(* CoDeSys 2.3.9.41 project: VOS_Vorkuta_ASU_1.pro *)
(* Libraries: GermesLib_1_51.lib 19.5.21 13:36:15, PID_Regulators.lib 6.11.19 15:29:27, Util.lib 18.5.10 15:14:28, STANDARD.LIB 4.10.05 11:14:46, IECSFC.LIB 13.4.06 15:51:28, SYSLIBTIME.LIB 6.11.19 15:29:28, ANALYZATION.LIB 5.10.99 09:05:06 *)

(* PLC configuration (modules and I/O channels)
Fast discrete inputs [I_SIMPLE_INPUT] node 0, in %IB0 out %QB0 {ChannellName = Fast discrete inputs; Filtrationtime = 10000}
  DD1_DI_1 AT %IX0.0 [BitInput] Discrete input 1 reserve {ChannellName = Enter name}
  DD1_DI_2 AT %IX0.1 [BitInput] Discrete input 2 reserve {ChannellName = Enter name}
  DD1_DI_3 AT %IX0.2 [BitInput] Discrete input 3 reserve {ChannellName = Enter name}
  DD1_DI_4 AT %IX0.3 [BitInput] Discrete input 4 reserve {ChannellName = Enter name}
Discrete inputs [ID130] node 1, in %IB1 out %QB1 {ChannellName = Discrete inputs; Filtrationtime_GeneralINP = 10; PinCount = 12; Visibility = No}
  AT %IB1.0 [ByteInput] 8 discrete inputs {ChannellName = Enter name}
  AT %IB1.1 [ByteInput] 4 discrete inputs {ChannellName = Enter name}
Fast discrete outputs [OWEN_ID570] node 2, in %IB2 out %QB2 {ChannellName = Fast discrete outputs; SafeValueBool = FALSE; SafeValueBool = FALSE; SafeValueBool = FALSE; SafeValueBool = FALSE; Visibility = No}
  AT %QX2.0 [BitOutput] Fast discrete output 1 {ChannellName = Enter name}
  AT %QX2.1 [BitOutput] Fast discrete output 2 {ChannellName = Enter name}
  AT %QX2.2 [BitOutput] Fast discrete output 3 {ChannellName = Enter name}
  AT %QX2.3 [BitOutput] Fast discrete output 4 {ChannellName = Enter name}
Discrete outputs [ID131] node 3, in %IB3 out %QB3 {ChannellName = Discrete outputs; SafeValueByte = 0; Visibility = No}
  AT %QB3.0 [ByteOutput] 8 discrete outputs {ChannellName = Enter name}
  AT %QB3.1 [ByteOutput] 8 discrete outputs {ChannellName = Enter name}
DD1_AI_1 AT %IR4.0 [FloatInputP] LT06.01/01 уровень в V06.01/01 {ChannellName = Fast analog input; AIN_TYPE = 0-20 mA; Peak_Filtr = 200; Flt_Ch = Off; TauRC = 10; MinFV = 0; MaxFV = 20000.0}
DD1_AI_2 AT %IR4.1 [FloatInputP] PT06.01/01 {ChannellName = Fast analog input; AIN_TYPE = 0-20 mA; Peak_Filtr = 200; Flt_Ch = Off; TauRC = 10; MinFV = 0; MaxFV = 20000.0}
DD1_AI_3 AT %IR4.2 [FloatInputP] PT06.01/02 {ChannellName = Fast analog input; AIN_TYPE = 0-20 mA; Peak_Filtr = 200; Flt_Ch = Off; TauRC = 10; MinFV = 0; MaxFV = 20000.0}
DD1_AI_4 AT %IR4.3 [FloatInputP] TT01.02 температура воздуха в помещении {ChannellName = Fast analog input; AIN_TYPE = 0-20 mA; Peak_Filtr = 200; Flt_Ch = Off; TauRC = 10; MinFV = 0; MaxFV = 20000.0}
DD1_AI_5 AT %IR4.4 [FloatInputP] TT06.01 температура воды на выходе {ChannellName = Fast analog input; AIN_TYPE = 0-20 mA; Peak_Filtr = 200; Flt_Ch = Off; TauRC = 10; MinFV = 0; MaxFV = 20000.0}
DD1_AI_6 AT %IR4.5 [FloatInputP] pH-метр QE06.01 {ChannellName = Fast analog input; AIN_TYPE = 0-20 mA; Peak_Filtr = 200; Flt_Ch = Off; TauRC = 10; MinFV = 0; MaxFV = 20000.0}
DD1_AI_7 AT %IR4.6 [FloatInputP] FIT06.01 расходомер на выходе {ChannellName = Fast analog input; AIN_TYPE = 0-20 mA; Peak_Filtr = 200; Flt_Ch = Off; TauRC = 10; MinFV = 0; MaxFV = 20000.0}
DD1_AI_8 AT %IR4.7 [FloatInputP] reserve {ChannellName = Fast analog input; AIN_TYPE = 0-20 mA; Peak_Filtr = 200; Flt_Ch = Off; TauRC = 10; MinFV = 0; MaxFV = 20000.0}
AT %IW4.8 [WordInput] AI read time (10ms) {ChannellName = Enter name}
Analog outputs [ID126] node 5, in %IB5 out %QB5 {ChannellName = Analog outputs}
  DD1_AO_1 AT %QR5.0 [FloatOutputP] производительность доз.насоса Р03.06/01 {ChannellName = Analog output; AOUT_TYPE = 4-20 mA; SafeValueREAL = 0.0}
  DD1_AO_2 AT %QR5.1 [FloatOutputP] производительность доз.насоса Р03.06/02 {ChannellName = Analog output; AOUT_TYPE = 4-20 mA; SafeValueREAL = 0.0}
  DD1_AO_3 AT %QR5.2 [FloatOutputP] reserve {ChannellName = Analog output; AOUT_TYPE = 4-20 mA; SafeValueREAL = 0.0}
  DD1_AO_4 AT %QR5.3 [FloatOutputP] reserve {ChannellName = Analog output; AOUT_TYPE = 4-20 mA; SafeValueREAL = 0.0}
Special input [ID103] node 6, in %IB6 out %QB6 {ChannellName = Special input}
  AT %IX6.0 [BitInput] Special input {ChannellName = Enter name}
Special output [ID104] node 7, in %IB7 out %QB7 {ChannellName = Special output}
  AT %QX7.0 [BitOutput] Special output {ChannellName = Enter name}
AT %QD8.0 [DWordOutput] Last address {ChannellName = Enter name}
AT %QW8.1 [WordOutput] Last error {ChannellName = Enter name}
RS-485-1 [COM1_USART] node 0, in %IB8.0 out %QB8.0 {ChannellName = RS-485-1; CommunicationSpeed = 115200; Parity = NO PARITY CHECK; BitLength = 8 bits; StopLength = One stop bit; InterfaceType = RS485; FrameOriented = RTU; Timeout = 2; Visibility = No}
Universal Modbus device [ID2000] node 1, in %IB8.1 out %QB8.1 {ChannellName = Universal Modbus device; ModuleIP = 10:0:0:223; ServiceTimeout = 150; TCPport = 502; NetMode = Serial; ModuleSlaveAddress = 11; RequestType = By poll time; PeriodOfService = 100; Visibility = No; RepeatCounter = 0; ByteSequence = Native}
  AT %QB8.1.0 [ComChannel] Command (0xff - Start) {ChannellName = Enter name}
  Real input module [ID2007] node 0, in %IB8.1.0 out %QB8.1.0 {ChannellName = float input module; ModbusAddress = 512; Command_read_regs = Read holding Registers  (0x03); Visibility = No}
    DD2_AI_1 AT %QD8.1.0.0 [FloatOutput] {ChannellName = Enter name}
  Real input module [ID2007] node 1, in %IB8.1.1 out %QB8.1.1 {ChannellName = float input module; ModbusAddress = 514; Command_read_regs = Read holding Registers  (0x03); Visibility = No}
    DD2_AI_2 AT %QD8.1.1.0 [FloatOutput] {ChannellName = Enter name}
  Real input module [ID2007] node 2, in %IB8.1.2 out %QB8.1.2 {ChannellName = float input module; ModbusAddress = 516; Command_read_regs = Read holding Registers  (0x03); Visibility = No}
    DD2_AI_3 AT %QD8.1.2.0 [FloatOutput] {ChannellName = Enter name}
  Real input module [ID2007] node 3, in %IB8.1.3 out %QB8.1.3 {ChannellName = float input module; ModbusAddress = 518; Command_read_regs = Read holding Registers  (0x03); Visibility = No}
    DD2_AI_4 AT %QD8.1.3.0 [FloatOutput] {ChannellName = Enter name}
  Real input module [ID2007] node 4, in %IB8.1.4 out %QB8.1.4 {ChannellName = float input module; ModbusAddress = 520; Command_read_regs = Read holding Registers  (0x03); Visibility = No}
    DD2_AI_5 AT %QD8.1.4.0 [FloatOutput] {ChannellName = Enter name}
  Real input module [ID2007] node 5, in %IB8.1.5 out %QB8.1.5 {ChannellName = float input module; ModbusAddress = 522; Command_read_regs = Read holding Registers  (0x03); Visibility = No}
    DD2_AI_6 AT %QD8.1.5.0 [FloatOutput] {ChannellName = Enter name}
  Real input module [ID2007] node 6, in %IB8.1.6 out %QB8.1.6 {ChannellName = float input module; ModbusAddress = 524; Command_read_regs = Read holding Registers  (0x03); Visibility = No}
    DD2_AI_7 AT %QD8.1.6.0 [FloatOutput] {ChannellName = Enter name}
  Real input module [ID2007] node 7, in %IB8.1.7 out %QB8.1.7 {ChannellName = float input module; ModbusAddress = 526; Command_read_regs = Read holding Registers  (0x03); Visibility = No}
    DD2_AI_8 AT %QD8.1.7.0 [FloatOutput] {ChannellName = Enter name}
  Register input module [ID2003] node 8, in %IB8.1.8 out %QB8.1.8 {ChannellName = Register input module; ModbusAddress = 528; Command_read_regs = Read input registers  (0x04); Visibility = No}
    DI_BitMask AT %QW8.1.8.0 [WordOutput] {ChannellName = Enter name}
  Register input module [ID2003] node 9, in %IB8.1.9 out %QB8.1.9 {ChannellName = Register input module; ModbusAddress = 531; Command_read_regs = Read input registers  (0x04); Visibility = No}
    stat_word_PLC_DD2 AT %QW8.1.9.0 [WordOutput] {ChannellName = Enter name}
Universal Modbus device [ID2000] node 2, in %IB8.2 out %QB8.2 {ChannellName = Universal Modbus device; ModuleIP = 10:0:0:223; ServiceTimeout = 150; TCPport = 502; NetMode = Serial; ModuleSlaveAddress = 12; RequestType = By poll time; PeriodOfService = 100; Visibility = No; RepeatCounter = 0; ByteSequence = Native}
  AT %QB8.2.0 [ComChannel] Command (0xff - Start) {ChannellName = Enter name}
  Real input module [ID2007] node 0, in %IB8.2.0 out %QB8.2.0 {ChannellName = float input module; ModbusAddress = 512; Command_read_regs = Read holding Registers  (0x03); Visibility = No}
    DD3_AI_1 AT %QD8.2.0.0 [FloatOutput] {ChannellName = Enter name}
  Real input module [ID2007] node 1, in %IB8.2.1 out %QB8.2.1 {ChannellName = float input module; ModbusAddress = 514; Command_read_regs = Read holding Registers  (0x03); Visibility = No}
    DD3_AI_2 AT %QD8.2.1.0 [FloatOutput] {ChannellName = Enter name}
  Register input module [ID2003] node 2, in %IB8.2.2 out %QB8.2.2 {ChannellName = Register input module; ModbusAddress = 516; Command_read_regs = Read input registers  (0x04); Visibility = No}
    stat_word_PLC_DD3 AT %QW8.2.2.0 [WordOutput] {ChannellName = Enter name}
  Register input module [ID2003] node 3, in %IB8.2.3 out %QB8.2.3 {ChannellName = Register input module; ModbusAddress = 518; Command_read_regs = Read input registers  (0x04); Visibility = No}
    stat_ufo_PLC AT %QW8.2.3.0 [WordOutput] {ChannellName = Enter name}
Universal Modbus device [ID2000] node 3, in %IB8.3 out %QB8.3 {ChannellName = Universal Modbus device; ModuleIP = 10:0:0:223; ServiceTimeout = 150; TCPport = 502; NetMode = Serial; ModuleSlaveAddress = 13; RequestType = By poll time; PeriodOfService = 100; Visibility = No; RepeatCounter = 0; ByteSequence = Trace_mode}
  AT %QB8.3.0 [ComChannel] Command (0xff - Start) {ChannellName = Enter name}
  Register input module [ID2003] node 0, in %IB8.3.0 out %QB8.3.0 {ChannellName = Register input module; ModbusAddress = 17; Command_read_regs = Read input registers  (0x04); Visibility = No}
    bitMask_DD4_DI AT %QW8.3.0.0 [WordOutput] {ChannellName = Enter name}
Universal Modbus device [ID2000] node 4, in %IB8.4 out %QB8.4 {ChannellName = Universal Modbus device; ModuleIP = 10:0:0:223; ServiceTimeout = 150; TCPport = 502; NetMode = Serial; ModuleSlaveAddress = 11; RequestType = By value change; PeriodOfService = 100; Visibility = No; RepeatCounter = 0; ByteSequence = Native}
  AT %QB8.4.0 [ComChannel] Command (0xff - Start) {ChannellName = Enter name}
  Register output module State [ID2014] node 0, in %IB8.4.0 out %QB8.4.0 {ChannellName = Register output module State; ModbusAddress = 529; Command_write_one_reg = Write multiple registers(0x10); Visibility = No}
    DO_BitMask AT %QW8.4.0.0 [WordOutput] {ChannellName = Enter name}
    AT %QB8.4.0.1 [ComChannel] Command (0xff - Start) {ChannellName = Enter name}
  Register output module State [ID2014] node 1, in %IB8.4.1 out %QB8.4.1 {ChannellName = Register output module State; ModbusAddress = 530; Command_write_one_reg = Write multiple registers(0x10); Visibility = No}
    com_word_PLC_DD2 AT %QW8.4.1.0 [WordOutput] {ChannellName = Enter name}
    AT %QB8.4.1.1 [ComChannel] Command (0xff - Start) {ChannellName = Enter name}
  Register output module [ID2004] node 2, in %IB8.4.2 out %QB8.4.2 {ChannellName = Register; ModbusAddress = 532; Command_write_one_reg = Write multiple registers(0x10); Visibility = No}
    set_freq_p010301_PLC AT %QW8.4.2.0 [WordOutput] {ChannellName = Enter name}
  Register output module [ID2004] node 3, in %IB8.4.3 out %QB8.4.3 {ChannellName = Register; ModbusAddress = 533; Command_write_one_reg = Write multiple registers(0x10); Visibility = No}
    set_freq_p010302_PLC AT %QW8.4.3.0 [WordOutput] {ChannellName = Enter name}
  Register output module [ID2004] node 4, in %IB8.4.4 out %QB8.4.4 {ChannellName = Register; ModbusAddress = 534; Command_write_one_reg = Write multiple registers(0x10); Visibility = No}
    set_freq_p010303_PLC AT %QW8.4.4.0 [WordOutput] {ChannellName = Enter name}
  Register output module [ID2004] node 5, in %IB8.4.5 out %QB8.4.5 {ChannellName = Register; ModbusAddress = 535; Command_write_one_reg = Write multiple registers(0x10); Visibility = No}
    set_freq_p010701_PLC AT %QW8.4.5.0 [WordOutput] {ChannellName = Enter name}
  Register output module [ID2004] node 6, in %IB8.4.6 out %QB8.4.6 {ChannellName = Register; ModbusAddress = 536; Command_write_one_reg = Write multiple registers(0x10); Visibility = No}
    set_freq_p010702_PLC AT %QW8.4.6.0 [WordOutput] {ChannellName = Enter name}
  Register output module [ID2004] node 7, in %IB8.4.7 out %QB8.4.7 {ChannellName = Register; ModbusAddress = 537; Command_write_one_reg = Write multiple registers(0x10); Visibility = No}
    set_freq_p010801_PLC AT %QW8.4.7.0 [WordOutput] {ChannellName = Enter name}
  Register output module [ID2004] node 8, in %IB8.4.8 out %QB8.4.8 {ChannellName = Register; ModbusAddress = 538; Command_write_one_reg = Write multiple registers(0x10); Visibility = No}
    set_freq_p010802_PLC AT %QW8.4.8.0 [WordOutput] {ChannellName = Enter name}
  Register output module [ID2004] node 9, in %IB8.4.9 out %QB8.4.9 {ChannellName = Register; ModbusAddress = 539; Command_write_one_reg = Write multiple registers(0x10); Visibility = No}
    set_freq_p060201_PLC AT %QW8.4.9.0 [WordOutput] {ChannellName = Enter name}
  Register output module [ID2004] node 10, in %IB8.4.10 out %QB8.4.10 {ChannellName = Register; ModbusAddress = 540; Command_write_one_reg = Write multiple registers(0x10); Visibility = No}
    set_freq_p060202_PLC AT %QW8.4.10.0 [WordOutput] {ChannellName = Enter name}
Universal Modbus device [ID2000] node 5, in %IB8.5 out %QB8.5 {ChannellName = Universal Modbus device; ModuleIP = 10:0:0:223; ServiceTimeout = 150; TCPport = 502; NetMode = Serial; ModuleSlaveAddress = 12; RequestType = By value change; PeriodOfService = 100; Visibility = No; RepeatCounter = 0; ByteSequence = Native}
  AT %QB8.5.0 [ComChannel] Command (0xff - Start) {ChannellName = Enter name}
  Register output module [ID2004] node 0, in %IB8.5.0 out %QB8.5.0 {ChannellName = Register; ModbusAddress = 517; Command_write_one_reg = Write multiple registers(0x10); Visibility = No}
    com_word_PLC_DD3 AT %QW8.5.0.0 [WordOutput] {ChannellName = Enter name}
*)

(* POU PLC_PRG, CFC *)
PROGRAM PLC_PRG
VAR
	P0103manager: RichThreePumpManager;
	TT0101rawValue: REAL;
	PT0101rawValue: REAL;
	PT0102rawValue: REAL;
	PT0103rawValue: REAL;
	LT0101rawValue: REAL;
	FIT0101rawValue: REAL;
	FIT0102rawValue: REAL;
	PH0101rawValue: REAL;
	alarmP010201: BOOL;
	alarmP010202: BOOL;
	alarmF0104power: BOOL;
	alarmValves1_9_23: BOOL;
	regenF010401: BOOL;
	alarmF010401: BOOL;
	regenF010402: BOOL;
	alarmF010402: BOOL;
	regenF010403: BOOL;
	alarmF010403: BOOL;
	highLevelV010501_LS0101: BOOL;
	midLevelV010501_LS0102: BOOL;
	lowLevelV010501_LS0103: BOOL;
	highLevelV070101_LS070101: BOOL;
	highLevelV011001_LS0105: BOOL;
	lowLevelV011001_LS0106: BOOL;
	valve1: BOOL;
	valve2: BOOL;
	valve3: BOOL;
	valve4: BOOL;
	valveReserve: BOOL;
	startP010201: BOOL;
	startP010202: BOOL;
	startRegenF010401: BOOL;
	startRegenF010402: BOOL;
	startRegenF010403: BOOL;
	reserveBool: BOOL;
	alarmP010301: BOOL;
	alarmP010302: BOOL;
	alarmP010303: BOOL;
	alarmP010701: BOOL;
	alarmP010702: BOOL;
	alarmP010801: BOOL;
	alarmP010802: BOOL;
	startP010301: BOOL;
	startP010302: BOOL;
	startP010303: BOOL;
	startP010701: BOOL;
	startP010702: BOOL;
	startP010801: BOOL;
	startP010802: BOOL;
	startP060201: BOOL;
	startP060202: BOOL;
	set_freq_p010301: UINT;
	set_freq_p010302: UINT;
	set_freq_p010303: UINT;
	set_freq_p010701: UINT;
	set_freq_p010702: UINT;
	set_freq_p010801: UINT;
	set_freq_p010802: UINT;
	set_freq_p060201: UINT;
	set_freq_p060202: UINT;
	PT0104rawValue: REAL;
	PT0105rawValue: REAL;
	resetAlarms: BOOL;
	startP080101: BOOL;
	startP080202: BOOL;
	startUFO1: BOOL;
	startUFO2: BOOL;
	stopUFO1: BOOL;
	stopUFO2: BOOL;
	alarmP050201: BOOL;
	alarmP050301: BOOL;
	alarmLowPIS0501: BOOL;
	alarmP080101: BOOL;
	alarmP080102: BOOL;
	highLevelV080101_LS0801: BOOL;
	lowLevelV080101_LS0802: BOOL;
	startedP050201: BOOL;
	startedP050301: BOOL;
	startedH050401: BOOL;
	heatingH050401: BOOL;

	UFO1_started: BOOL;
	UFO1_overheatDecontaminationCamera: BOOL;
	UFO1_overheatControlPanel: BOOL;
	UFO1_alarmLamp: BOOL;
	UFO1_alarmControlPanel: BOOL;
	UFO1_warning_lowUF: BOOL;
	UFO1_alarm_lowUF: BOOL;
	UFO1_alarm_UFsensor: BOOL;

	UFO2_started: BOOL;
	UFO2_overheatDecontaminationCamera: BOOL;
	UFO2_overheatControlPanel: BOOL;
	UFO2_alarmLamp: BOOL;
	UFO2_alarmControlPanel: BOOL;
	UFO2_warning_lowUF: BOOL;
	UFO2_alarm_lowUF: BOOL;
	UFO2_alarm_UFsensor: BOOL;
	highLevelV0109_LS0104: BOOL;		(*кондуктометрический датчик верхнего уровня в обезвоживателе*)
	alarmP060301: BOOL;
	alarmP060302: BOOL;
	startP060301: BOOL;
	startP060302: BOOL;
	LT060101rawValue: REAL;
	PT060101rawValue: REAL;
	PT060102rawValue: REAL;
	TT0102rawValue: REAL;
	TT0601rawValue: REAL;
	PH0601rawValue: REAL;
	FIT0601rawValue: REAL;
	setCapacityP060301: REAL;		(*задать производительность доз.насоса Р06.03/01*)
	setCapacityP060302: REAL;		(*задать производительность доз.насоса Р06.03/02*)
	CAI_1: ControlAI;
	CAI_2: ControlAI;
	CAI_3: ControlAI;
	CAI_4: ControlAI;
	CAI_5: ControlAI;
	CAI_6: ControlAI;
	CAI_7: ControlAI;
	CAI_8: ControlAI;
	CAI_9: ControlAI;
	CAI_10: ControlAI;
	CAI_11: ControlAI;
	CAI_12: ControlAI;
	CAI_13: ControlAI;
	CAI_14: ControlAI;
	CAI_15: ControlAI;
	CAI_16: ControlAI;
	CAI_17: ControlAI;

	alarmLT060101: BOOL;		(*авария датчика РТ06.01/01*)
	alarmPT060101: BOOL;		(*авария датчика РТ06.01/01*)
	alarmPT060102: BOOL;
	alarmTT0102: BOOL;
	alarmTT0601: BOOL;
	alarmPH0601: BOOL;
	alarmFIT0601: BOOL;
	alarmTT0101: BOOL;
	alarmPT0101: BOOL;
	alarmPT0102: BOOL;
	alarmPT0103: BOOL;
	alarmLT0101: BOOL;
	alarmFIT0101: BOOL;
	alarmFIT0102: BOOL;
	alarmPH0101: BOOL;
	alarmPT0104: BOOL;
	alarmPT0105: BOOL;

	LT060101realValue: REAL;		(*реальная физическая величина по показаниям датчика*)
	PT060101realValue: REAL;
	PT060102realValue: REAL;
	TT0102realValue: REAL;
	TT0601realValue: REAL;
	PH0601realValue: REAL;
	FIT0601realValue: REAL;
	TT0101realValue: REAL;
	PT0101realValue: REAL;
	PT0102realValue: REAL;
	PT0103realValue: REAL;
	LT0101realValue: REAL;
	FIT0101realValue: REAL;
	FIT0102realValue: REAL;
	PH0101realValue: REAL;
	PT0104realValue: REAL;
	PT0105realValue: REAL;
END_VAR
VAR RETAIN
	LT060101maxValue: REAL;		(*max физическая величина соответствующая 20мА*)
	PT060101maxValue: REAL;
	PT060102maxValue: REAL;
	TT0102maxValue: REAL;
	TT0601maxValue: REAL;
	PH0601maxValue: REAL;
	FIT0601maxValue: REAL;
	TT0101maxValue: REAL;
	PT0101maxValue: REAL;
	PT0102maxValue: REAL;
	PT0103maxValue: REAL;
	LT0101maxValue: REAL;
	FIT0101maxValue: REAL;
	FIT0102maxValue: REAL;
	PH0101maxValue: REAL;
	PT0104maxValue: REAL;
	PT0105maxValue: REAL;
END_VAR
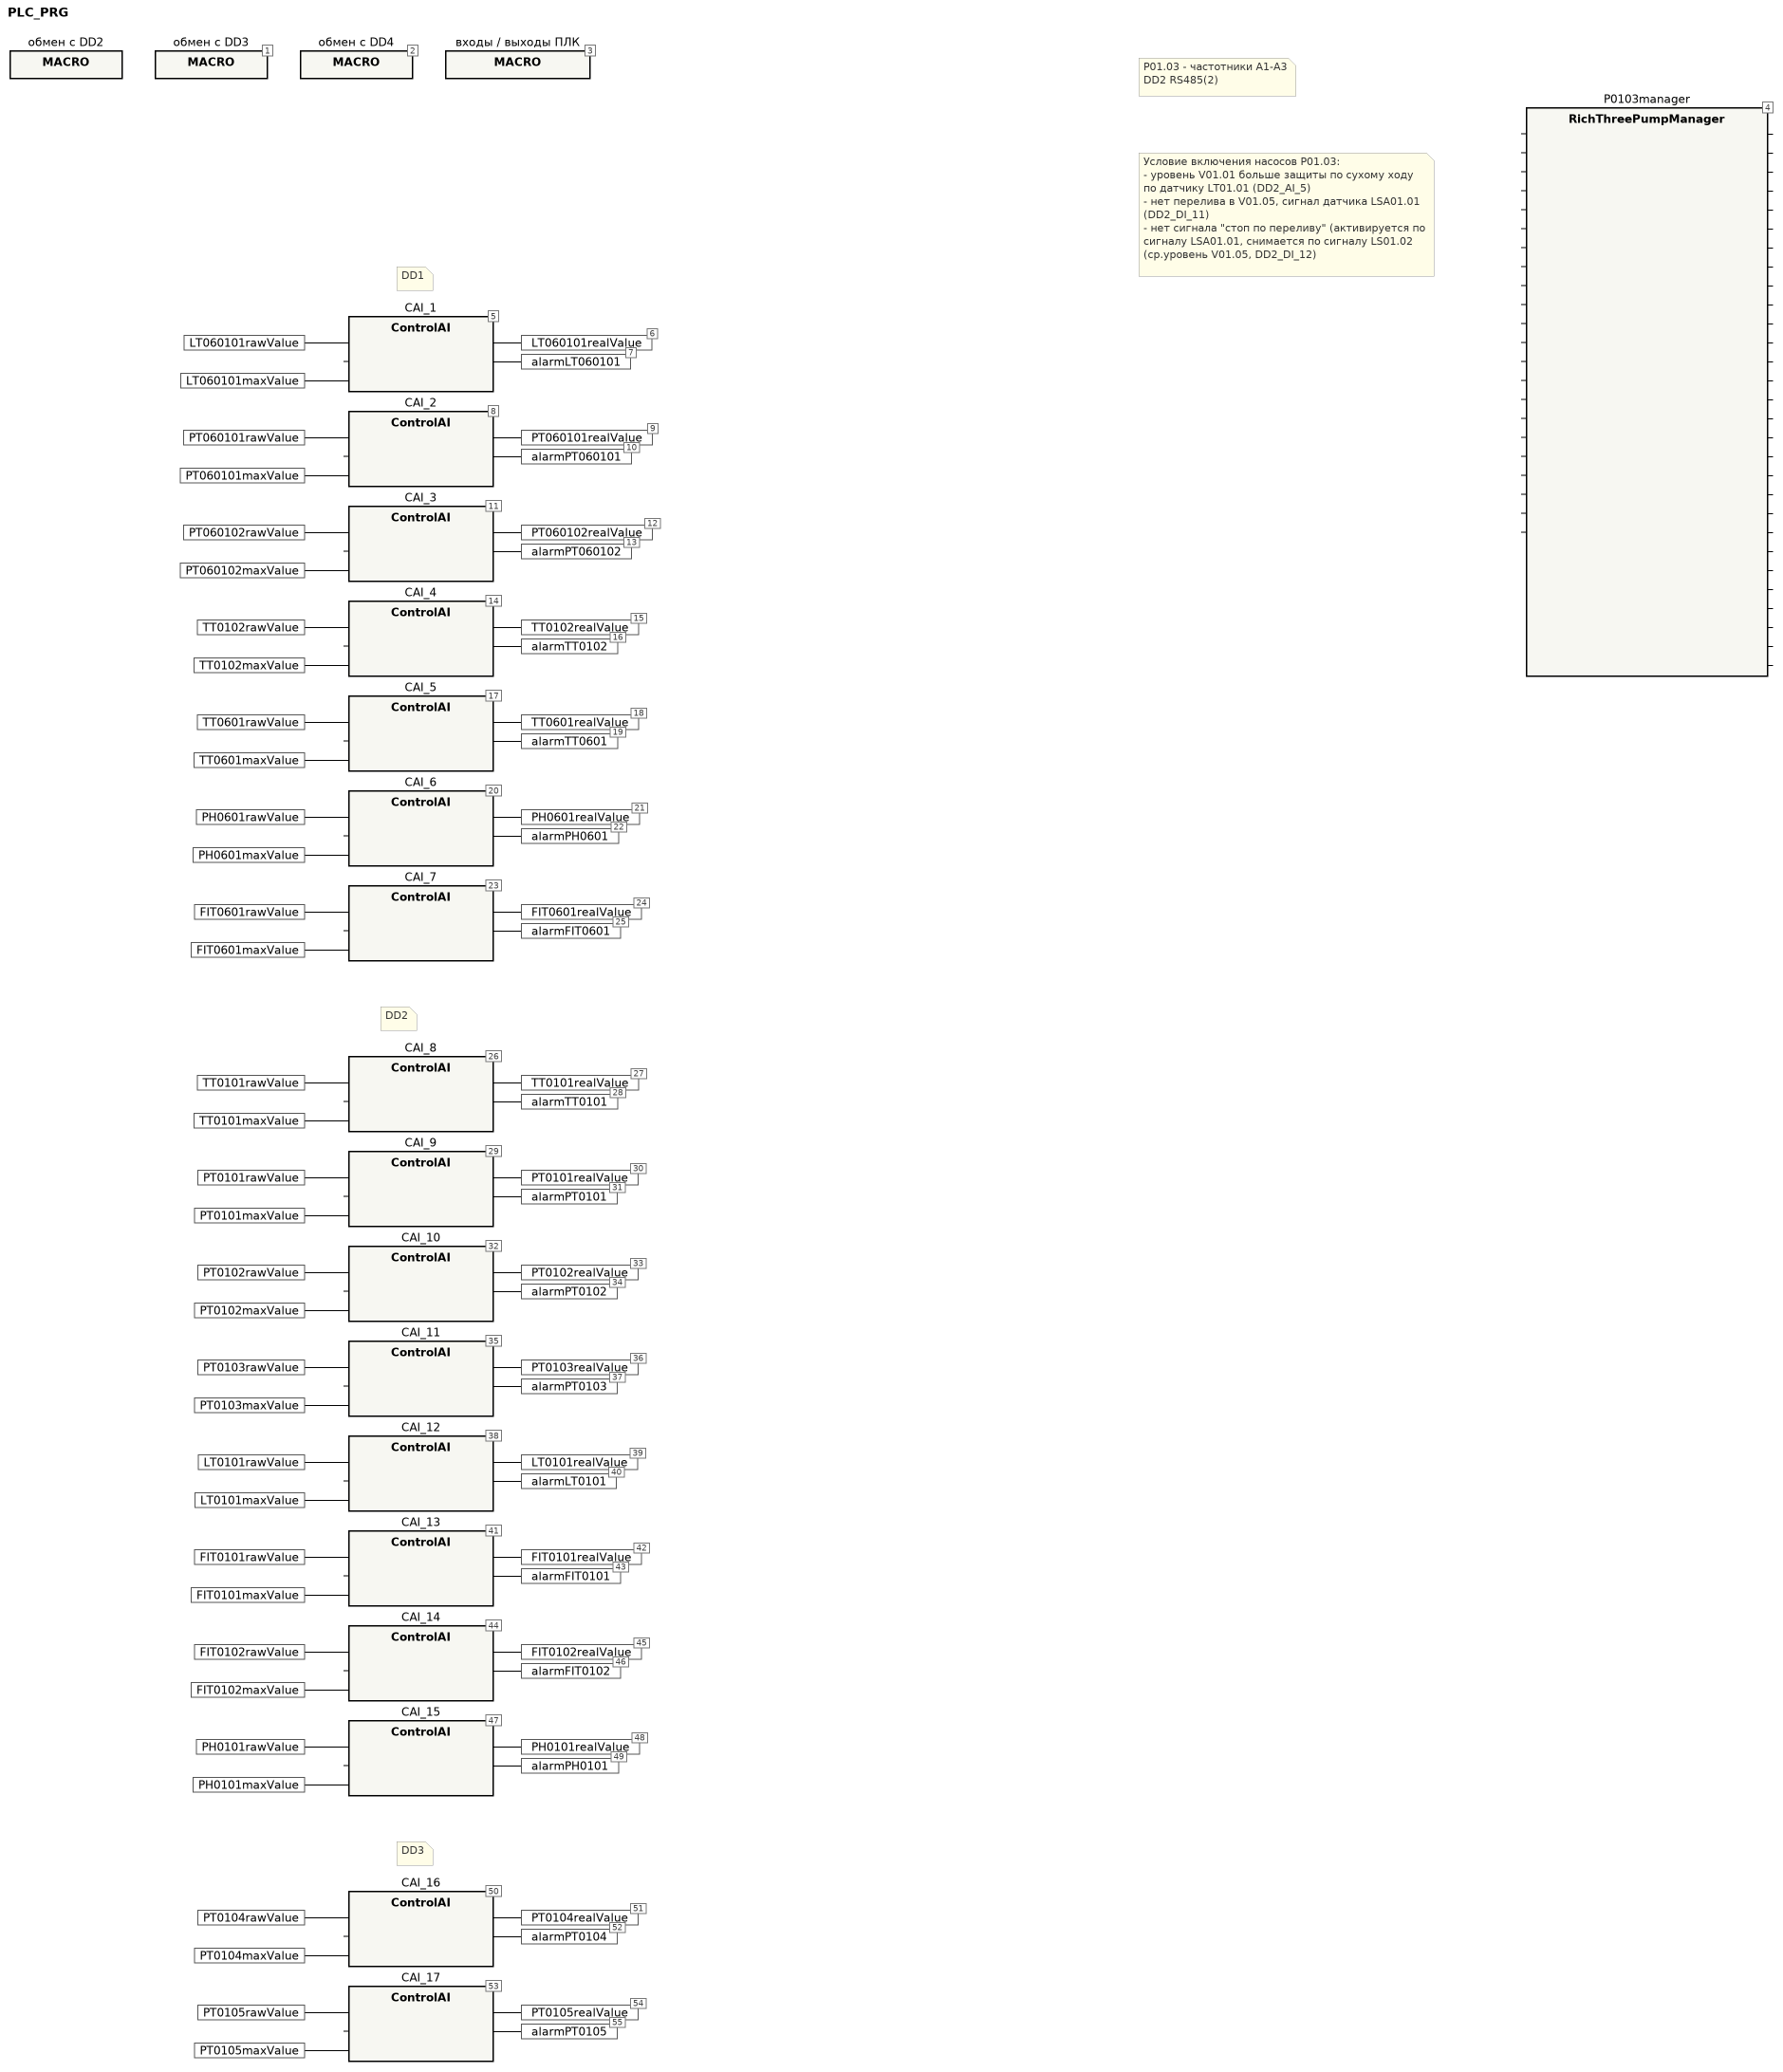
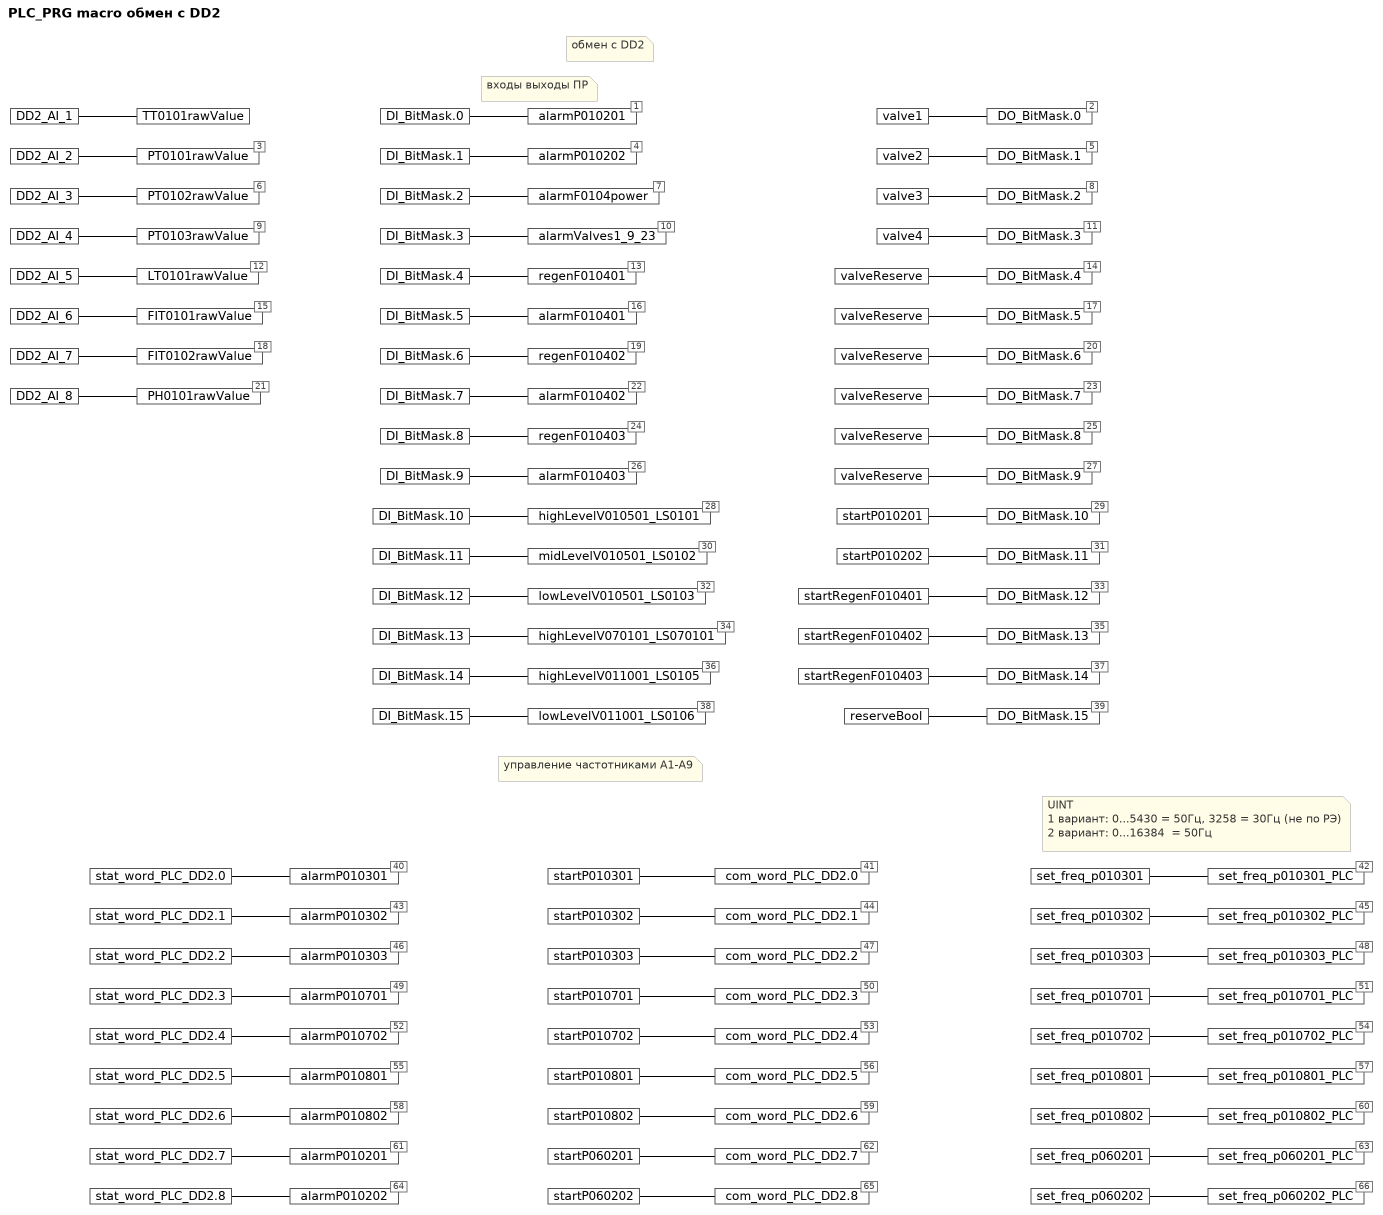
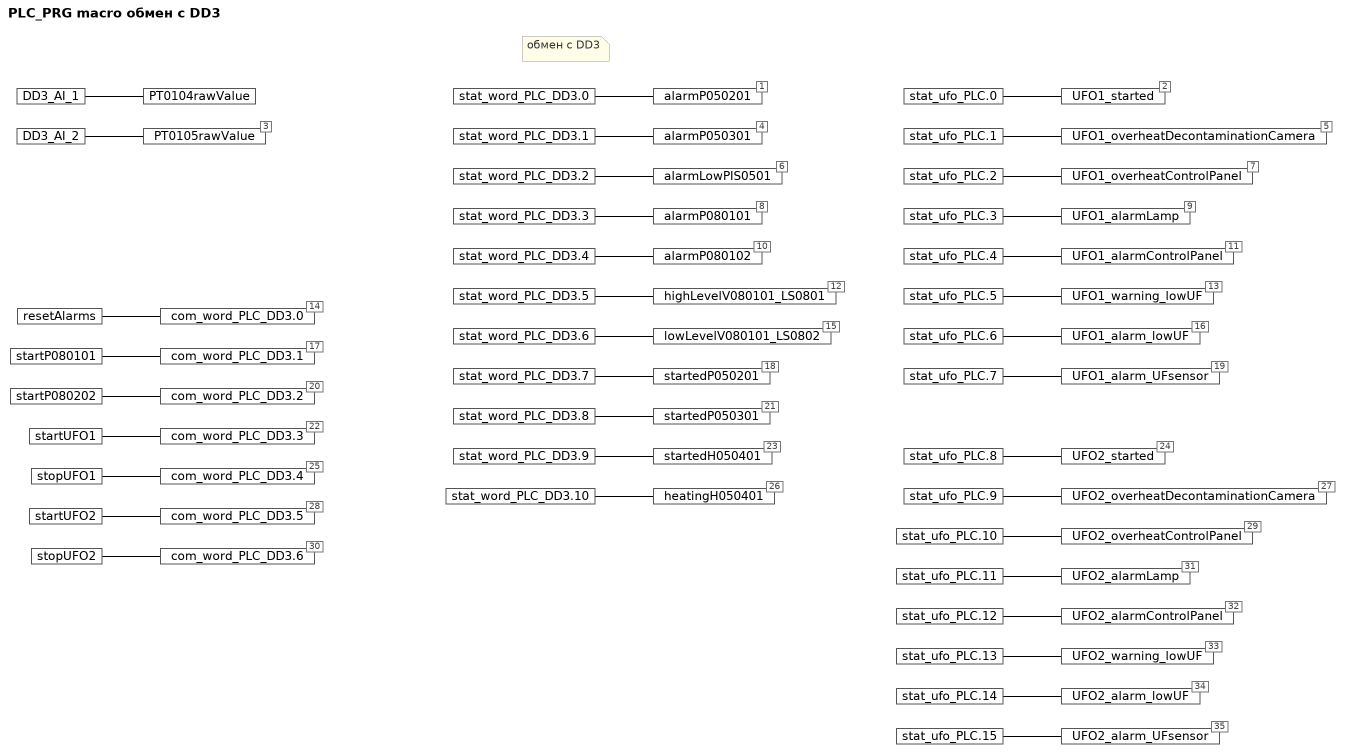
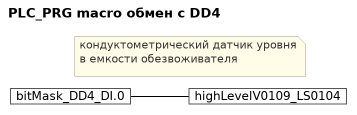
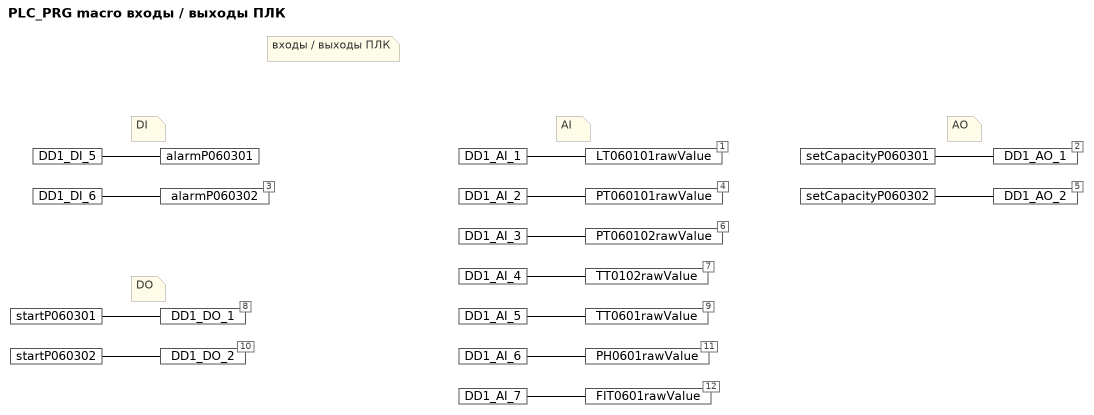
_CFC_ (* Continuous Function Chart, elements in execution order *)
(* DD2 *)
(* DD3 *)
(* DD1 *)
(* P01.03 - частотники А1-А3 / DD2 RS485(2) *)
(* Условие включения насосов Р01.03: / - уровень V01.01 больше защиты по сухому ходу / по датчику LT01.01 (DD2_AI_5) / - нет перелива в V01.05, сигнал датчика LSA01.01 / (DD2_DI_11) / - нет сигнала "стоп по переливу" (активируется по / сигналу LSA01.01, снимается по сигналу LS01.02 / (ср.уровень V01.05, DD2_DI_12) *)
#0 MACRO обмен с DD2()
	(* UINT / 1 вариант: 0...5430 = 50Гц, 3258 = 30Гц (не по РЭ) / 2 вариант: 0...16384  = 50Гц *)
	(* обмен с DD2 *)
	(* входы выходы ПР *)
	(* управление частотниками А1-А9 *)
	#1 TT0101rawValue <= DD2_AI_1
	#2 alarmP010201 <= DI_BitMask.0
	#3 DO_BitMask.0 <= valve1
	#4 PT0101rawValue <= DD2_AI_2
	#5 alarmP010202 <= DI_BitMask.1
	#6 DO_BitMask.1 <= valve2
	#7 PT0102rawValue <= DD2_AI_3
	#8 alarmF0104power <= DI_BitMask.2
	#9 DO_BitMask.2 <= valve3
	#10 PT0103rawValue <= DD2_AI_4
	#11 alarmValves1_9_23 <= DI_BitMask.3
	#12 DO_BitMask.3 <= valve4
	#13 LT0101rawValue <= DD2_AI_5
	#14 regenF010401 <= DI_BitMask.4
	#15 DO_BitMask.4 <= valveReserve
	#16 FIT0101rawValue <= DD2_AI_6
	#17 alarmF010401 <= DI_BitMask.5
	#18 DO_BitMask.5 <= valveReserve
	#19 FIT0102rawValue <= DD2_AI_7
	#20 regenF010402 <= DI_BitMask.6
	#21 DO_BitMask.6 <= valveReserve
	#22 PH0101rawValue <= DD2_AI_8
	#23 alarmF010402 <= DI_BitMask.7
	#24 DO_BitMask.7 <= valveReserve
	#25 regenF010403 <= DI_BitMask.8
	#26 DO_BitMask.8 <= valveReserve
	#27 alarmF010403 <= DI_BitMask.9
	#28 DO_BitMask.9 <= valveReserve
	#29 highLevelV010501_LS0101 <= DI_BitMask.10
	#30 DO_BitMask.10 <= startP010201
	#31 midLevelV010501_LS0102 <= DI_BitMask.11
	#32 DO_BitMask.11 <= startP010202
	#33 lowLevelV010501_LS0103 <= DI_BitMask.12
	#34 DO_BitMask.12 <= startRegenF010401
	#35 highLevelV070101_LS070101 <= DI_BitMask.13
	#36 DO_BitMask.13 <= startRegenF010402
	#37 highLevelV011001_LS0105 <= DI_BitMask.14
	#38 DO_BitMask.14 <= startRegenF010403
	#39 lowLevelV011001_LS0106 <= DI_BitMask.15
	#40 DO_BitMask.15 <= reserveBool
	#41 alarmP010301 <= stat_word_PLC_DD2.0
	#42 com_word_PLC_DD2.0 <= startP010301
	#43 set_freq_p010301_PLC <= set_freq_p010301
	#44 alarmP010302 <= stat_word_PLC_DD2.1
	#45 com_word_PLC_DD2.1 <= startP010302
	#46 set_freq_p010302_PLC <= set_freq_p010302
	#47 alarmP010303 <= stat_word_PLC_DD2.2
	#48 com_word_PLC_DD2.2 <= startP010303
	#49 set_freq_p010303_PLC <= set_freq_p010303
	#50 alarmP010701 <= stat_word_PLC_DD2.3
	#51 com_word_PLC_DD2.3 <= startP010701
	#52 set_freq_p010701_PLC <= set_freq_p010701
	#53 alarmP010702 <= stat_word_PLC_DD2.4
	#54 com_word_PLC_DD2.4 <= startP010702
	#55 set_freq_p010702_PLC <= set_freq_p010702
	#56 alarmP010801 <= stat_word_PLC_DD2.5
	#57 com_word_PLC_DD2.5 <= startP010801
	#58 set_freq_p010801_PLC <= set_freq_p010801
	#59 alarmP010802 <= stat_word_PLC_DD2.6
	#60 com_word_PLC_DD2.6 <= startP010802
	#61 set_freq_p010802_PLC <= set_freq_p010802
	#62 alarmP010201 <= stat_word_PLC_DD2.7
	#63 com_word_PLC_DD2.7 <= startP060201
	#64 set_freq_p060201_PLC <= set_freq_p060201
	#65 alarmP010202 <= stat_word_PLC_DD2.8
	#66 com_word_PLC_DD2.8 <= startP060202
	#67 set_freq_p060202_PLC <= set_freq_p060202
END_MACRO
#68 MACRO обмен с DD3()
	(* обмен с DD3 *)
	#69 PT0104rawValue <= DD3_AI_1
	#70 alarmP050201 <= stat_word_PLC_DD3.0
	#71 UFO1_started <= stat_ufo_PLC.0
	#72 PT0105rawValue <= DD3_AI_2
	#73 alarmP050301 <= stat_word_PLC_DD3.1
	#74 UFO1_overheatDecontaminationCamera <= stat_ufo_PLC.1
	#75 alarmLowPIS0501 <= stat_word_PLC_DD3.2
	#76 UFO1_overheatControlPanel <= stat_ufo_PLC.2
	#77 alarmP080101 <= stat_word_PLC_DD3.3
	#78 UFO1_alarmLamp <= stat_ufo_PLC.3
	#79 alarmP080102 <= stat_word_PLC_DD3.4
	#80 UFO1_alarmControlPanel <= stat_ufo_PLC.4
	#81 highLevelV080101_LS0801 <= stat_word_PLC_DD3.5
	#82 UFO1_warning_lowUF <= stat_ufo_PLC.5
	#83 com_word_PLC_DD3.0 <= resetAlarms
	#84 lowLevelV080101_LS0802 <= stat_word_PLC_DD3.6
	#85 UFO1_alarm_lowUF <= stat_ufo_PLC.6
	#86 com_word_PLC_DD3.1 <= startP080101
	#87 startedP050201 <= stat_word_PLC_DD3.7
	#88 UFO1_alarm_UFsensor <= stat_ufo_PLC.7
	#89 com_word_PLC_DD3.2 <= startP080202
	#90 startedP050301 <= stat_word_PLC_DD3.8
	#91 com_word_PLC_DD3.3 <= startUFO1
	#92 startedH050401 <= stat_word_PLC_DD3.9
	#93 UFO2_started <= stat_ufo_PLC.8
	#94 com_word_PLC_DD3.4 <= stopUFO1
	#95 heatingH050401 <= stat_word_PLC_DD3.10
	#96 UFO2_overheatDecontaminationCamera <= stat_ufo_PLC.9
	#97 com_word_PLC_DD3.5 <= startUFO2
	#98 UFO2_overheatControlPanel <= stat_ufo_PLC.10
	#99 com_word_PLC_DD3.6 <= stopUFO2
	#100 UFO2_alarmLamp <= stat_ufo_PLC.11
	#101 UFO2_alarmControlPanel <= stat_ufo_PLC.12
	#102 UFO2_warning_lowUF <= stat_ufo_PLC.13
	#103 UFO2_alarm_lowUF <= stat_ufo_PLC.14
	#104 UFO2_alarm_UFsensor <= stat_ufo_PLC.15
END_MACRO
#105 MACRO обмен с DD4()
	(* кондуктометрический датчик уровня / в емкости обезвоживателя *)
	#106 highLevelV0109_LS0104 <= bitMask_DD4_DI.0
END_MACRO
#107 MACRO входы / выходы ПЛК()
	(* AI *)
	(* DO *)
	(* DI *)
	(* входы / выходы ПЛК *)
	(* AO *)
	#108 alarmP060301 <= DD1_DI_5
	#109 LT060101rawValue <= DD1_AI_1
	#110 DD1_AO_1 <= setCapacityP060301
	#111 alarmP060302 <= DD1_DI_6
	#112 PT060101rawValue <= DD1_AI_2
	#113 DD1_AO_2 <= setCapacityP060302
	#114 PT060102rawValue <= DD1_AI_3
	#115 TT0102rawValue <= DD1_AI_4
	#116 DD1_DO_1 <= startP060301
	#117 TT0601rawValue <= DD1_AI_5
	#118 DD1_DO_2 <= startP060302
	#119 PH0601rawValue <= DD1_AI_6
	#120 FIT0601rawValue <= DD1_AI_7
END_MACRO
#121 P0103manager:RichThreePumpManager(-, -, -, -, -, -, -, -, -, -, -, -, -, -, -, -, -, -, -, -, -, -)
#122 CAI_1:ControlAI(LT060101rawValue, -, LT060101maxValue)
#123 LT060101realValue <= #122.out 1
#124 alarmLT060101 <= #122.out 2
#125 CAI_2:ControlAI(PT060101rawValue, -, PT060101maxValue)
#126 PT060101realValue <= #125.out 1
#127 alarmPT060101 <= #125.out 2
#128 CAI_3:ControlAI(PT060102rawValue, -, PT060102maxValue)
#129 PT060102realValue <= #128.out 1
#130 alarmPT060102 <= #128.out 2
#131 CAI_4:ControlAI(TT0102rawValue, -, TT0102maxValue)
#132 TT0102realValue <= #131.out 1
#133 alarmTT0102 <= #131.out 2
#134 CAI_5:ControlAI(TT0601rawValue, -, TT0601maxValue)
#135 TT0601realValue <= #134.out 1
#136 alarmTT0601 <= #134.out 2
#137 CAI_6:ControlAI(PH0601rawValue, -, PH0601maxValue)
#138 PH0601realValue <= #137.out 1
#139 alarmPH0601 <= #137.out 2
#140 CAI_7:ControlAI(FIT0601rawValue, -, FIT0601maxValue)
#141 FIT0601realValue <= #140.out 1
#142 alarmFIT0601 <= #140.out 2
#143 CAI_8:ControlAI(TT0101rawValue, -, TT0101maxValue)
#144 TT0101realValue <= #143.out 1
#145 alarmTT0101 <= #143.out 2
#146 CAI_9:ControlAI(PT0101rawValue, -, PT0101maxValue)
#147 PT0101realValue <= #146.out 1
#148 alarmPT0101 <= #146.out 2
#149 CAI_10:ControlAI(PT0102rawValue, -, PT0102maxValue)
#150 PT0102realValue <= #149.out 1
#151 alarmPT0102 <= #149.out 2
#152 CAI_11:ControlAI(PT0103rawValue, -, PT0103maxValue)
#153 PT0103realValue <= #152.out 1
#154 alarmPT0103 <= #152.out 2
#155 CAI_12:ControlAI(LT0101rawValue, -, LT0101maxValue)
#156 LT0101realValue <= #155.out 1
#157 alarmLT0101 <= #155.out 2
#158 CAI_13:ControlAI(FIT0101rawValue, -, FIT0101maxValue)
#159 FIT0101realValue <= #158.out 1
#160 alarmFIT0101 <= #158.out 2
#161 CAI_14:ControlAI(FIT0102rawValue, -, FIT0102maxValue)
#162 FIT0102realValue <= #161.out 1
#163 alarmFIT0102 <= #161.out 2
#164 CAI_15:ControlAI(PH0101rawValue, -, PH0101maxValue)
#165 PH0101realValue <= #164.out 1
#166 alarmPH0101 <= #164.out 2
#167 CAI_16:ControlAI(PT0104rawValue, -, PT0104maxValue)
#168 PT0104realValue <= #167.out 1
#169 alarmPT0104 <= #167.out 2
#170 CAI_17:ControlAI(PT0105rawValue, -, PT0105maxValue)
#171 PT0105realValue <= #170.out 1
#172 alarmPT0105 <= #170.out 2
_END_CFC_
END_PROGRAM
